# EPICS substitutions: apps/svtApp/Db/crate.substitutions
# SVT HFCB HV & LV wiener modules substitution file
#
#  for iseg (HV) MX is slot # 1-10
file iocsoftsvtAppsV/db/iseg.db {
pattern { HOST, MX }
  {"vmetlsvt1","7"}
  {"vmetlsvt1","8"}
  {"vmetlsvt1","9"}
  {"vmetlsvt1","10"}
  {"vmetlsvt4","8"}
  {"vmetlsvt4","9"}
  {"vmetlsvt4","10"}
}
#  for mpv (LV) MX is slot # 0-9
file iocsoftsvtAppsV/db/mpv.db {
   pattern { HOST, MX }
  {"vmetlsvt1","0"}
  {"vmetlsvt1","1"}
  {"vmetlsvt1","2"}
  {"vmetlsvt1","3"}
  {"vmetlsvt1","4"}
  {"vmetlsvt4","0"}
  {"vmetlsvt4","1"}
  {"vmetlsvt4","2"}
  {"vmetlsvt4","3"}
  {"vmetlsvt4","4"}
  {"vmetlsvt4","5"}
  {"vmetlsvt4","6"}
}
